PROGRAM MAIN
VAR
END_VAR

RESTFUL_API();

END_PROGRAM

(* stored: Version 1.1.0.1, ProductVersion 3.1.4024.13
   POU MAIN: Id {0c102052-944a-4d15-b53d-3e28cc8fcd91}, SpecialFunc None *)
